FUNCTION_BLOCK InterpretarComando
VAR_INPUT
END_VAR
VAR_OUTPUT
END_VAR
VAR
	aux_str:STRING;
	aux_int:INT;
	aux_real:REAL;
END_VAR

IF IO.ready THEN

	IF  LEFT(IO.string_in, 1)='G' THEN
		IF LEFT(IO.string_in, 3) ='G00' THEN
			IO.string_out:='comando G00 recibido';
			//buscar comandos de X
			IF FIND (IO.string_in,'X') > 0 THEN
			aux_int:=FIND (IO.string_in,'X');
			aux_str:=MID(IO.string_in,3,aux_int+1);
			aux_real:=STRING_TO_REAL(aux_str);
			GVL.Xc_sp:= aux_real;
			GVL.comando_actual:=IO.string_in;
			IO.ready:=FALSE;
			END_IF
			//buscar comandos de Y
			IF FIND (IO.string_in,'Y') > 0 THEN
			aux_int:=FIND (IO.string_in,'Y');
			aux_str:=MID(IO.string_in,3,aux_int+1);
			aux_real:=STRING_TO_REAL(aux_str);
			GVL.Yc_sp:= aux_real;
			GVL.comando_actual:=IO.string_in;
			IO.ready:=FALSE;
			END_IF
			
		END_IF
		ELSE IF LEFT(IO.string_in, 3) ='G01' THEN
			IO.string_out:='comando G01 recibido';
			GVL.comando_actual:=IO.string_in;
	ELSE IO.string_out:='Comando desconocido';
		GVL.comando_actual:='Comando desconocido';
		IO.ready:=TRUE;
	END_IF
END_IF
END_IF

END_FUNCTION_BLOCK

(* stored: Version 1.1.0.1, ProductVersion 3.1.4024.4
   POU InterpretarComando: Id {c6ae15c2-f634-45d8-9d77-e1f929492264}, SpecialFunc None *)
